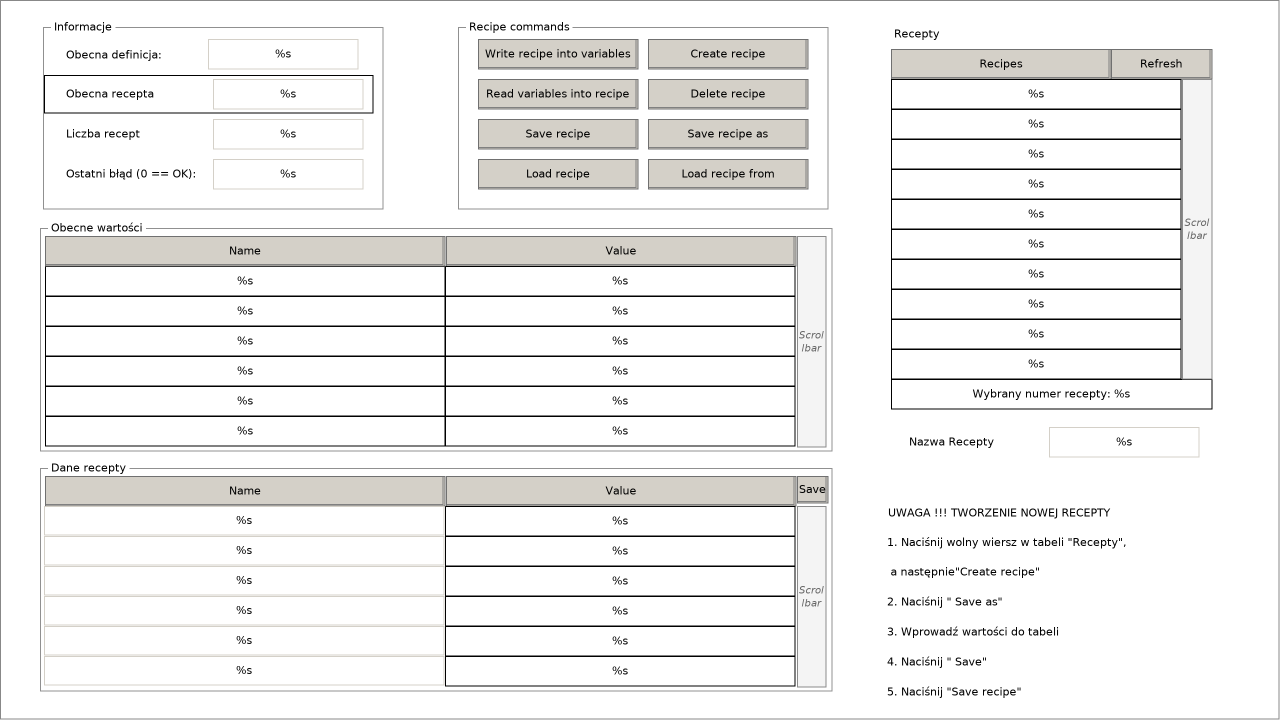
VISUALIZATION Visualization  // 1280x720
    GroupBox (40,220 792x231), "Obecne wartości"
        Rectangle (5,46 400x30), "%s", text variable: GVL_RecipeTable.aVariableNames[GVL_RecipeTable.nVariableIndex], input disabled if: TRUE
        Rectangle (5,76 400x30), "%s", text variable: GVL_RecipeTable.aVariableNames[GVL_RecipeTable.nVariableIndex+1], input disabled if: TRUE
        Rectangle (5,136 400x30), "%s", text variable: GVL_RecipeTable.aVariableNames[GVL_RecipeTable.nVariableIndex+3], input disabled if: TRUE
        Rectangle (5,166 400x30), "%s", text variable: GVL_RecipeTable.aVariableNames[GVL_RecipeTable.nVariableIndex+4], input disabled if: TRUE
        Rectangle (5,196 400x30), "%s", text variable: GVL_RecipeTable.aVariableNames[GVL_RecipeTable.nVariableIndex+5], input disabled if: TRUE
        Rectangle (5,106 400x30), "%s", text variable: GVL_RecipeTable.aVariableNames[GVL_RecipeTable.nVariableIndex+2], input disabled if: TRUE
    GroupBox (40,460 792x231), "Dane recepty"
    GroupBox (43,19 340x190), "Informacje"
        Rectangle (1,56 329x38)
        Textfield (165,20 150x30), "%s", text variable: RecipeManagement.sRecipeDef, input disabled if: TRUE
            OnMouseClick: write the text variable via Default
        Label (20,21 150x30), "Obecna definicja:"
        Label (20,60 150x30), "Obecna recepta"
        Label (20,140 150x30), "Ostatni błąd (0 == OK):"
        Label (20,100 150x30), "Liczba recept"
        Textfield (170,60 150x30), "%s", text variable: RecipeManagement.sRecipe, input disabled if: TRUE
            OnMouseClick: write the text variable via Default
        Textfield (170,140 150x30), "%s", text variable: RecipeManagement.nLastError, input disabled if: TRUE
        Textfield (170,100 150x30), "%s", text variable: RecipeManagement.nRecipeCount, input disabled if: TRUE
    GroupBox (458,19 370x190), "Recipe commands"
        Button (20,20 160x30), "Write recipe into variables"
            OnMouseClick: ExecuteCommand ExecuteCommand=ExecuteCommand=[Command=WriteRecipe, Value=RecipeManagement.sRecipeDef, Value2=RecipeManagement.sRecipe]
        Button (20,60 160x30), "Read variables into recipe"
            OnMouseClick: ExecuteCommand ExecuteCommand=ExecuteCommand=[Command=ReadRecipe, Value=RecipeManagement.sRecipeDef, Value2=RecipeManagement.sRecipe]
            OnMouseClick: execute { RecipeManagement.bReloadValues := TRUE; }
        Button (20,100 160x30), "Save recipe"
            OnMouseClick: ExecuteCommand ExecuteCommand=ExecuteCommand=[Command=SaveRecipe, Value=RecipeManagement.sRecipeDef, Value2=RecipeManagement.sRecipe]
        Button (20,140 160x30), "Load recipe"
            OnMouseClick: ExecuteCommand ExecuteCommand=ExecuteCommand=[Command=LoadRecipe, Value=RecipeManagement.sRecipeDef, Value2=RecipeManagement.sRecipe]
            OnMouseClick: toggle RecipeManagement.bReloadValues
            OnMouseClick: execute {
                GVL_RecipeTable.aCurrentValues[0]:=GVL_Recipe.dl_kartonu;
                GVL_RecipeTable.aCurrentValues[1]:=GVL_Recipe.wys_kartonu;
                GVL_RecipeTable.aCurrentValues[2]:=GVL_Recipe.szer_kartonu;
                GVL_RecipeTable.aCurrentValues[3]:=GVL_Recipe.Poz_X_Odlozenie;
                GVL_RecipeTable.aCurrentValues[4]:=GVL_Recipe.Il_kolumn;
                GVL_RecipeTable.aCurrentValues[5]:=GVL_Recipe.Il_rzedow;
                GVL_RecipeTable.aCurrentValues[6]:=GVL_Recipe.Predk_mag_odlozenie;
                GVL_RecipeTable.aCurrentValues[7]:=GVL_Recipe.Predk_mag_pobranie;
                GVL_RecipeTable.aCurrentValues[8]:=GVL_Recipe.Predk_plot_odlozenie;
                GVL_RecipeTable.aCurrentValues[9]:=GVL_Recipe.Predk_plot_pobranie;
                GVL_RecipeTable.aCurrentValues[10]:=GVL_Recipe.Predk_plot_ruch;
                GVL_RecipeTable.aCurrentValues[11]:=GVL_Recipe.Poz_Z_Odlozenie;
                GVL_RecipeTable.aCurrentValues[12]:=GVL_Recipe.Poz_Z_Pobranie;
            }
            OnMouseClick: execute { GVL_RecipeTable.aCurrentVariableNames:=GVL_RecipeTable.aVariableNames; }
        Button (190,20 160x30), "Create recipe"
            OnMouseClick: ExecuteCommand ExecuteCommand=ExecuteCommand=[Command=CreateRecipe, Value=RecipeManagement.sRecipeDef, Value2=MAIN.sRecipe]
            OnMouseClick: execute { RecipeManagement.bReload := TRUE; }
        Button (190,100 160x30), "Save recipe as"
            OnMouseClick: ExecuteCommand ExecuteCommand=ExecuteCommand=[Command=SaveRecipeAs, Value=RecipeManagement.sRecipeDef, Value2=RecipeManagement.sRecipe]
        Button (190,140 160x30), "Load recipe from"
            OnMouseClick: ExecuteCommand ExecuteCommand=ExecuteCommand=[Command=LoadRecipeFrom, Value=RecipeManagement.sRecipeDef, Value2=RecipeManagement.sRecipe]
        Button (190,60 160x30), "Delete recipe"
            OnMouseClick: ExecuteCommand ExecuteCommand=ExecuteCommand=[Command=DeleteRecipe, Value=RecipeManagement.sRecipeDef, Value2=RecipeManagement.sRecipe]
            OnMouseClick: execute { RecipeManagement.bInit := TRUE; }
    Button (891,49 220x30), "Recipes"
        OnMouseDown: toggle RecipeManagement.bReload
    Label (891,19 322x30), "Recepty"
    Button (1111,49 101x30), "Refresh"
        OnMouseDown: toggle RecipeManagement.bReload
    Rectangle (891,79 290x30), "%s", text variable: GVL_RecipeTable.aRecipeNames[GVL_RecipeTable.nRecipeIndex], colour toggle: (GVL_RecipeTable.nRecipeSelectionIndex-GVL_RecipeTable.nRecipeIndex) = 0
        OnMouseDown: execute { GVL_RecipeTable.nRecipeSelectionIndex := GVL_RecipeTable.nRecipeIndex; }
    Rectangle (891,109 290x30), "%s", text variable: GVL_RecipeTable.aRecipeNames[GVL_RecipeTable.nRecipeIndex+1], colour toggle: (GVL_RecipeTable.nRecipeSelectionIndex-GVL_RecipeTable.nRecipeIndex) = 1
        OnMouseDown: execute { GVL_RecipeTable.nRecipeSelectionIndex := GVL_RecipeTable.nRecipeIndex + 1; }
    Rectangle (891,139 290x30), "%s", text variable: GVL_RecipeTable.aRecipeNames[GVL_RecipeTable.nRecipeIndex+2], colour toggle: (GVL_RecipeTable.nRecipeSelectionIndex-GVL_RecipeTable.nRecipeIndex) = 2
        OnMouseDown: execute { GVL_RecipeTable.nRecipeSelectionIndex := GVL_RecipeTable.nRecipeIndex + 2; }
    Rectangle (891,169 290x30), "%s", text variable: GVL_RecipeTable.aRecipeNames[GVL_RecipeTable.nRecipeIndex+3], colour toggle: (GVL_RecipeTable.nRecipeSelectionIndex-GVL_RecipeTable.nRecipeIndex) = 3
        OnMouseDown: execute { GVL_RecipeTable.nRecipeSelectionIndex := GVL_RecipeTable.nRecipeIndex + 3; }
    Rectangle (891,199 290x30), "%s", text variable: GVL_RecipeTable.aRecipeNames[GVL_RecipeTable.nRecipeIndex+4], colour toggle: (GVL_RecipeTable.nRecipeSelectionIndex-GVL_RecipeTable.nRecipeIndex) = 4
        OnMouseDown: execute { GVL_RecipeTable.nRecipeSelectionIndex := GVL_RecipeTable.nRecipeIndex + 4; }
    Rectangle (891,229 290x30), "%s", text variable: GVL_RecipeTable.aRecipeNames[GVL_RecipeTable.nRecipeIndex+5], colour toggle: (GVL_RecipeTable.nRecipeSelectionIndex-GVL_RecipeTable.nRecipeIndex) = 5
        OnMouseDown: execute { GVL_RecipeTable.nRecipeSelectionIndex := GVL_RecipeTable.nRecipeIndex + 5; }
    Rectangle (891,259 290x30), "%s", text variable: GVL_RecipeTable.aRecipeNames[GVL_RecipeTable.nRecipeIndex+6], colour toggle: (GVL_RecipeTable.nRecipeSelectionIndex-GVL_RecipeTable.nRecipeIndex) = 6
        OnMouseDown: execute { GVL_RecipeTable.nRecipeSelectionIndex := GVL_RecipeTable.nRecipeIndex + 6; }
    Rectangle (891,289 290x30), "%s", text variable: GVL_RecipeTable.aRecipeNames[GVL_RecipeTable.nRecipeIndex+7], colour toggle: (GVL_RecipeTable.nRecipeSelectionIndex-GVL_RecipeTable.nRecipeIndex) = 7
        OnMouseDown: execute { GVL_RecipeTable.nRecipeSelectionIndex := GVL_RecipeTable.nRecipeIndex + 7; }
    Rectangle (891,319 290x30), "%s", text variable: GVL_RecipeTable.aRecipeNames[GVL_RecipeTable.nRecipeIndex+8], colour toggle: (GVL_RecipeTable.nRecipeSelectionIndex-GVL_RecipeTable.nRecipeIndex) = 8
        OnMouseDown: execute { GVL_RecipeTable.nRecipeSelectionIndex := GVL_RecipeTable.nRecipeIndex + 8; }
    Rectangle (891,349 290x30), "%s", text variable: GVL_RecipeTable.aRecipeNames[GVL_RecipeTable.nRecipeIndex+9], colour toggle: (GVL_RecipeTable.nRecipeSelectionIndex-GVL_RecipeTable.nRecipeIndex) = 9
        OnMouseDown: execute { GVL_RecipeTable.nRecipeSelectionIndex := GVL_RecipeTable.nRecipeIndex + 9; }
    Rectangle (891,379 321x30), "Wybrany numer recepty: %s", text variable: GVL_RecipeTable.nRecipeSelectionIndex+1, input disabled if: TRUE
    Scrollbar (1182,79 30x300)
        p2245068023: GVL_RecipeTable.nRecipeCount
        p1057716461: GVL_RecipeTable.nRecipeIndex
    Group (884,498 321x209)
        Label (0,29 321x31), "1. Naciśnij wolny wiersz w tabeli "Recepty","
        Label (1,0 271x30), "UWAGA !!! TWORZENIE NOWEJ RECEPTY"
        Label (0,59 150x30), "a następnie"Create recipe""
        Label (0,149 150x30), "4. Naciśnij " Save""
        Label (0,89 150x30), "2. Naciśnij " Save as""
        Label (0,179 150x30)
        Label (0,119 183x30), "3. Wprowadź wartości do tabeli"
        Label (0,179 150x30), "5. Naciśnij "Save recipe""
    Button (446,476 350x30), "Value"
    Button (797,476 31x27), "Save"
        OnMouseDown: toggle RecipeManagement.bSaveVariables
    Rectangle (445,506 350x30), "%s", text variable: GVL_RecipeTable.aVariableValues[GVL_RecipeTable.nVariableIndex]
        OnMouseDown: write the text variable via Edit
    Rectangle (445,536 350x30), "%s", text variable: GVL_RecipeTable.aVariableValues[GVL_RecipeTable.nVariableIndex+1]
        OnMouseDown: write the text variable via Edit
    Rectangle (445,566 350x30), "%s", text variable: GVL_RecipeTable.aVariableValues[GVL_RecipeTable.nVariableIndex+2]
        OnMouseDown: write the text variable via Edit
    Rectangle (445,596 350x30), "%s", text variable: GVL_RecipeTable.aVariableValues[GVL_RecipeTable.nVariableIndex+3]
        OnMouseDown: write the text variable via Edit
    Rectangle (445,626 350x30), "%s", text variable: GVL_RecipeTable.aVariableValues[GVL_RecipeTable.nVariableIndex+4]
        OnMouseDown: write the text variable via Edit
    Scrollbar (797,506 29x181)
        p1057716461: GVL_RecipeTable.nVariableIndex
    Rectangle (445,656 350x30), "%s", text variable: GVL_RecipeTable.aVariableValues[GVL_RecipeTable.nVariableIndex+5]
        OnMouseDown: write the text variable via Edit
    Button (45,476 400x30), "Name"
    Textfield (44,506 400x29), "%s", text variable: GVL_RecipeTable.aVariableNames[GVL_RecipeTable.nVariableIndex], input disabled if: TRUE
        OnMouseClick: write the text variable via Default
    Textfield (44,536 400x29), "%s", text variable: GVL_RecipeTable.aVariableNames[GVL_RecipeTable.nVariableIndex+1], input disabled if: TRUE
        OnMouseClick: write the text variable via Default
    Textfield (44,566 400x29), "%s", text variable: GVL_RecipeTable.aVariableNames[GVL_RecipeTable.nVariableIndex+2], input disabled if: TRUE
        OnMouseClick: write the text variable via Default
    Textfield (44,596 400x29), "%s", text variable: GVL_RecipeTable.aVariableNames[GVL_RecipeTable.nVariableIndex+3], input disabled if: TRUE
        OnMouseClick: write the text variable via Default
    Textfield (44,626 400x29), "%s", text variable: GVL_RecipeTable.aVariableNames[GVL_RecipeTable.nVariableIndex+4], input disabled if: TRUE
        OnMouseClick: write the text variable via Default
    Textfield (44,656 400x29), "%s", text variable: GVL_RecipeTable.aVariableNames[GVL_RecipeTable.nVariableIndex+5], input disabled if: TRUE
        OnMouseClick: write the text variable via Default
    Button (446,236 350x30), "Value"
    Rectangle (445,266 350x30), "%s", text variable: GVL_RecipeTable.aCurrentValues[GVL_RecipeTable.nVariableIndex], input disabled if: TRUE
        OnMouseDown: write the text variable via Edit
    Rectangle (445,296 350x30), "%s", text variable: GVL_RecipeTable.aCurrentValues[GVL_RecipeTable.nVariableIndex+1], input disabled if: TRUE
        OnMouseDown: write the text variable via Edit
    Rectangle (445,326 350x30), "%s", text variable: GVL_RecipeTable.aCurrentValues[GVL_RecipeTable.nVariableIndex+2], input disabled if: TRUE
        OnMouseDown: write the text variable via Edit
    Rectangle (445,356 350x30), "%s", text variable: GVL_RecipeTable.aCurrentValues[GVL_RecipeTable.nVariableIndex+3], input disabled if: TRUE
        OnMouseDown: write the text variable via Edit
    Rectangle (445,386 350x30), "%s", text variable: GVL_RecipeTable.aCurrentValues[GVL_RecipeTable.nVariableIndex+4], input disabled if: TRUE
        OnMouseDown: write the text variable via Edit
    Scrollbar (797,236 29x211)
        p1057716461: GVL_RecipeTable.nVariableIndex1
    Rectangle (445,416 350x30), "%s", text variable: GVL_RecipeTable.aCurrentValues[GVL_RecipeTable.nVariableIndex+5], input disabled if: TRUE
        OnMouseDown: write the text variable via Edit
    Button (45,236 400x30), "Name"
    Label (906,427 150x30), "Nazwa Recepty"
    Textfield (1049,427 150x30), "%s", text variable: MAIN.sRecipe
END_VISUALIZATION

(* stored: Version 1.1.0.1, ProductVersion 3.1.4022.12
   Visu Visualization: Id {7c80b83f-eb0f-4e0e-baee-9070c17c89b8} *)
